{attribute 'GeneratedUsingTerminal: EPP1816-3008-0016'}
{attribute addProperty BoxType "EPP1816-3008-0016"}
{attribute addProperty Id "ErrorBOOL1TxPDO_ToggleBOOL1"}
{attribute addProperty CRC "2745852447"}
{attribute addProperty Size "2"}
TYPE Status_A3AA621F :
STRUCT
	{attribute addProperty Name "Error"}
	Error : BOOL;
	{attribute addProperty Name "TxPDO_Toggle"}
	TxPDO_Toggle : BOOL;
END_STRUCT
END_TYPE

(* stored: Version 1.2.0.0, ProductVersion 3.1.4024.9
   DUT Status_A3AA621F: Id {9d3f3d2c-402f-4427-a93a-2b050ccacdd2} *)
